// Mitsubishi GX Works2 project: 231002-001- exercicios-1   PLC: Q03UDV

// task Task_01 (event TRUE, interval 0, priority 31): POU_01

PROGRAM POU_01
(* structured ladder/FBD written out as ST: instructions are called as NAME(EN, inputs, outputs); _pN, _eN, _tN stand for wires *)
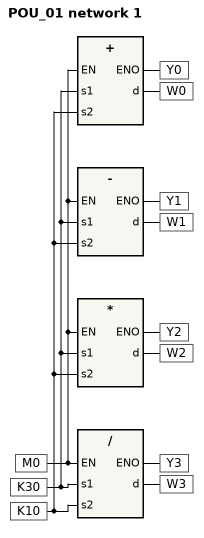
(* network 1 *)
_e1 := +(M0, K30, K10, W0);
Y0 := _e1;
_e2 := -(M0, K30, K10, W1);
Y1 := _e2;
_e3 := *(M0, K30, K10, W2);
Y2 := _e3;
_e4 := /(M0, K30, K10, W3);
Y3 := _e4;
END_PROGRAM
